Yaskawa INFORM job: BUFFER_WAIT.JBI

/JOB
//NAME BUFFER_WAIT
//POS
///NPOS 0,0,0,0,0,0
//INST
///DATE 2011/12/08 13:27
///ATTR SC,RW
///GROUP1 RB1
NOP
WHILE I091>I092
	 TIMER T=0.01
ENDWHILE
INC I091
END
